// TIA Portal V19 export
FUNCTION "FC10_Vacuum" : Void   // FC10, LAD
{ S7_Optimized_Access := 'TRUE' }
// stored: AutoNumber false, IsIECCheckEnabled true, SetENOAutomatically false
BEGIN

REGION Network 1: Complet management of Vacuum system
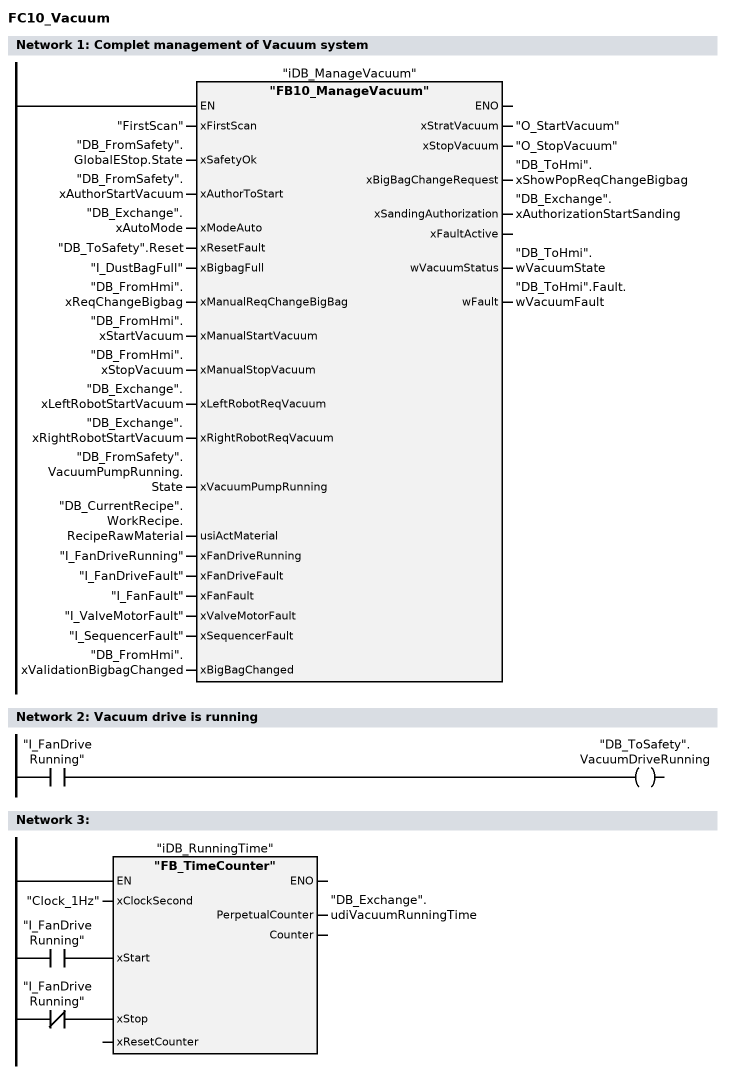
   RUNG wire#powerrail
      "iDB_ManageVacuum"(xFirstScan := "FirstScan", xSafetyOk := "DB_FromSafety".GlobalEStop.State, xAuthorToStart := "DB_FromSafety".xAuthorStartVacuum, xModeAuto := "DB_Exchange".xAutoMode, xResetFault := "DB_ToSafety".Reset, xBigbagFull := "I_DustBagFull", xManualReqChangeBigBag := "DB_FromHmi".xReqChangeBigbag, xManualStartVacuum := "DB_FromHmi".xStartVacuum, xManualStopVacuum := "DB_FromHmi".xStopVacuum, xLeftRobotReqVacuum := "DB_Exchange".xLeftRobotStartVacuum, xRightRobotReqVacuum := "DB_Exchange".xRightRobotStartVacuum, xVacuumPumpRunning := "DB_FromSafety".VacuumPumpRunning.State, usiActMaterial := "DB_CurrentRecipe".WorkRecipe.RecipeRawMaterial, xFanDriveRunning := "I_FanDriveRunning", xFanDriveFault := "I_FanDriveFault", xFanFault := "I_FanFault", xValveMotorFault := "I_ValveMotorFault", xSequencerFault := "I_SequencerFault", xBigBagChanged := "DB_FromHmi".xValidationBigbagChanged, xStratVacuum => "O_StartVacuum", xStopVacuum => "O_StopVacuum", xBigBagChangeRequest => "DB_ToHmi".xShowPopReqChangeBigbag, xSandingAuthorization => "DB_Exchange".xAuthorizationStartSanding, xFaultActive =>, wVacuumStatus => "DB_ToHmi".wVacuumState, wFault => "DB_ToHmi".Fault.wVacuumFault)
   END_RUNG
   // the same network as SCL:
   "iDB_ManageVacuum"(xFirstScan := "FirstScan",   // "FB10_ManageVacuum"
                      xSafetyOk := "DB_FromSafety".GlobalEStop.State,
                      xAuthorToStart := "DB_FromSafety".xAuthorStartVacuum,
                      xModeAuto := "DB_Exchange".xAutoMode,
                      xResetFault := "DB_ToSafety".Reset,
                      xBigbagFull := "I_DustBagFull",
                      xManualReqChangeBigBag := "DB_FromHmi".xReqChangeBigbag,
                      xManualStartVacuum := "DB_FromHmi".xStartVacuum,
                      xManualStopVacuum := "DB_FromHmi".xStopVacuum,
                      xLeftRobotReqVacuum := "DB_Exchange".xLeftRobotStartVacuum,
                      xRightRobotReqVacuum := "DB_Exchange".xRightRobotStartVacuum,
                      xVacuumPumpRunning := "DB_FromSafety".VacuumPumpRunning.State,
                      usiActMaterial := "DB_CurrentRecipe".WorkRecipe.RecipeRawMaterial,
                      xFanDriveRunning := "I_FanDriveRunning",
                      xFanDriveFault := "I_FanDriveFault",
                      xFanFault := "I_FanFault",
                      xValveMotorFault := "I_ValveMotorFault",
                      xSequencerFault := "I_SequencerFault",
                      xBigBagChanged := "DB_FromHmi".xValidationBigbagChanged,
                      xStratVacuum => "O_StartVacuum",
                      xStopVacuum => "O_StopVacuum",
                      xBigBagChangeRequest => "DB_ToHmi".xShowPopReqChangeBigbag,
                      xSandingAuthorization => "DB_Exchange".xAuthorizationStartSanding,
                      wVacuumStatus => "DB_ToHmi".wVacuumState,
                      wFault => "DB_ToHmi".Fault.wVacuumFault);
END_REGION

REGION Network 2: Vacuum drive is running
   RUNG wire#powerrail
      Contact( "I_FanDriveRunning" )
      Coil( "DB_ToSafety".VacuumDriveRunning )
   END_RUNG
   // the same network as SCL:
   "DB_ToSafety".VacuumDriveRunning := "I_FanDriveRunning";
END_REGION

REGION Network 3
   RUNG wire#powerrail
      "iDB_RunningTime"(xStart := wire#w1, xStop := wire#w2, xClockSecond := "Clock_1Hz", xResetCounter :=, PerpetualCounter => "DB_Exchange".udiVacuumRunningTime, "Counter" =>)
   END_RUNG
   RUNG wire#powerrail
      Contact( "I_FanDriveRunning" )
   END_RUNG wire#w1
   RUNG wire#powerrail
      I_Contact( "I_FanDriveRunning" )
   END_RUNG wire#w2
   // the same network as SCL:
   "iDB_RunningTime"(xClockSecond := "Clock_1Hz",   // "FB_TimeCounter"
                     xStart := "I_FanDriveRunning",
                     xStop := NOT "I_FanDriveRunning",
                     PerpetualCounter => "DB_Exchange".udiVacuumRunningTime);
END_REGION
END_FUNCTION
